(* PLC project Generated.project, CODESYS CODESYS V3.5 SP19 Patch 1 *)
(* stored: creationDateTime 2026-11-18T13:29:44.072454, modificationDateTime 2026-11-18T13:29:44.072454 *)

(* ======================================================================= 🧭 ST_MachineHoming — Etat publie du homing conjoint machine (M1/M2/benne) ─────────────────────────────────────────────────────────────── 🎯 Rôle : Regroupe les 8 sorties homing a plat de PRG_02_Acquisition en un bus struct unique, publie sur le bus inter-PRG. 🔒 Sécurité : Homed = qualification conjointe reference machine (gate SEMI_AUTO). HomingLoss = perte reference en mouvement : arret controle SafeStop. 📄 Doc métier : DOC/AF/AF_Partie-09_Fonction_Encoder_v2.4.md (F09.08) ======================================================================= *)
TYPE ST_MachineHoming : STRUCT
  Homed : BOOL;  (* Qualification conjointe reference machine *)
  SetPosBucketOpen : BOOL;  (* Valider position actuelle = reference benne ouverte *)
  SetPosBucketClose : BOOL;  (* Valider position actuelle = reference benne fermee *)
  Active : BOOL;  (* Homing conjoint en cours *)
  HomingLoss : BOOL;  (* Perte reference en mouvement : arret controle SafeStop *)
  Step : INT;  (* Etape guidee reference (echelle de priorite E_MachineHomingStep) *)
  Instruction : STRING(120);  (* Consigne IHM reference *)
  Failed : BOOL;  (* Transaction reference abandonnee *)
  SeqStep : INT;  (* Step GRAFCET courant (E_MachineHomingTxState HX0..HXF) *)
  M3Locked : BOOL;  (* Translation M3 interdite pendant le cycle de homing machine *)
  CmdWinchM1 : ST_ProgramWinchRequest;  (* Ordre treuil M1 couple palier 1 (HX2 montee / HX3 descente) *)
  CmdWinchM2 : ST_ProgramWinchRequest;  (* Ordre treuil M2 couple palier 1 (HX2 montee / HX3 descente) *)
  CmdBucketOpen : BOOL;  (* Ordre ouverture benne palier 1 sans FDC soft *)
  CmdBucketClose : BOOL;  (* Ordre fermeture benne palier 1 sans FDC soft (HX1) *)
  CmdWinchSelect : INT;  (* Override selecteur treuil cycle homing (-1=neutre, 0=couple, 2=benne) *)
  AllowAscent : BOOL;  (* Autorisation montee par etape GRAFCET homing *)
  AllowDescend : BOOL;  (* Autorisation descente par etape GRAFCET homing *)
  SoftLimitsOff : BOOL;  (* Inhibition limites soft position (HX1..HX3 uniquement, hors capteur TOP) *)
  BucketRefInvalidate : BOOL;  (* Revoque reference benne sur abandon cycle avant HX4 *)
  ProvisionalActive : BOOL;  (* TRUE tant que le zero 0m HX1 est provisoire avant HX4 8.5m *)
  TopContactLatched : BOOL;  (* Contact TOP touche pendant cycle homing : degagement requis *)
  TopContactCount : UINT;  (* Nombre de contacts capteur TOP pendant cycle homing (purge Reset) *)
  ActionText : STRING(120);  (* Consigne d action directe du GRAFCET pour bandeau operateur *)
END_STRUCT;
END_TYPE

(* ======================================================================= 🔌 ST_ProgramWinchRequest — Demande de mouvement treuil par le programme ─────────────────────────────────────────────────────────────── 🎯 Rôle : Regroupe les demandes logiques de treuil formulées par le séquenceur 📄 Référentiel : DOC/WFLOW/CONTRACTS/INTERPRG_CONTRACT_PRG03_MODES_CYCLE_v1.0.md ======================================================================= *)
TYPE ST_ProgramWinchRequest : STRUCT
  RunRequest : BOOL;  (* Ordre marche demandé par le programme *)
  ReqAscent : BOOL;  (* Demande montée *)
  ReqDescend : BOOL;  (* Demande descente *)
  StepTgt : INT;  (* Palier de vitesse cible demandé (1 à 5, 0 = arrêt) *)
END_STRUCT;
END_TYPE
